// TIA Portal V19 export
FUNCTION "FC_Korbumlaeufe" : Void   // FC330, LAD
TITLE = Korbumläufe
{ S7_Optimized_Access := 'TRUE' }
// stored: AutoNumber false, SetENOAutomatically false
   VAR_INPUT
      Nr : USInt;
   END_VAR
BEGIN

REGION Network 1 (SCL): Check Korb-Nr
   IF (#Nr < "KorbAnzahl_min") OR (#Nr > "KorbAnzahl_max") THEN
       RETURN;
   END_IF;
END_REGION

REGION Network 2 (SCL): Zählen und Maxwert checken
   "DB_Korbumlaeufe".Korb[#Nr].Durchlaeufe := "DB_Korbumlaeufe".Korb[#Nr].Durchlaeufe + 1;
END_REGION
END_FUNCTION
